FUNCTION_BLOCK VECTOR_DOT_P (* Dot product between two vector *)
  (* Standard: 61499-2 *)
  (* Version 1.0, 02-05-12, GASR, Universidade do Estado de Santa Catarina *)
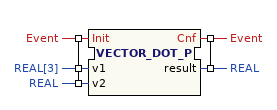
  EVENT_INPUT
    Init WITH v1, v2;
  END_EVENT
  EVENT_OUTPUT
    Cnf WITH result;
  END_EVENT
  VAR_INPUT
    v1 : ARRAY [0..2] OF REAL;
    v2 : REAL;
  END_VAR
  VAR_OUTPUT
    result : REAL;
  END_VAR
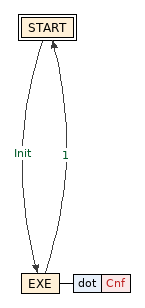
  EC_STATES
    START;
    EXE : dot -> Cnf;
  END_STATES
  EC_TRANSITIONS
    START TO EXE := Init;
    EXE TO START := 1;
  END_TRANSITIONS
  ALGORITHM dot IN Lua:
for i = 1, 3 do
        result = result + v1[ i ]*v2[ i ]
end
  END_ALGORITHM
END_FUNCTION_BLOCK
